{attribute 'GeneratedUsingTerminal: EK1122-0000-0018'}
{attribute addProperty BoxType "EK1122-0000-0018"}
{attribute addProperty Id "Beckhoff_ER6xxxsub_EK1100EK1100_AB5A94672A_0001_ER6001_0002_0016ER6001_B965E9F560A_0002_ER6001_0002_0021ER6001_B965E9F560A_0003_ER6002_0002_0021ER6002_EA7A2404108A_0004_ER6002_0002_0022ER6002_EECF1379108A_0005_ER6002_0002_0023ER6002_EECF1379108"}
{attribute addProperty CRC "2923937941"}
{attribute addProperty Size "446"}
TYPE Beckhoff_ER6xxxEK1122_AE47C095 EXTENDS EK1122_AB5A9467 :
STRUCT
	{attribute addProperty Name "Beckhoff_ER6xxxsub_EK1100"}
	{attribute addProperty PreviousPort "Beckhoff ER6xxxEK1122 : D"}
	Beckhoff_ER6xxxsub_EK1100 : EK1100_AB5A9467;
	{attribute addProperty Name "A_0001_ER6001_0002_0016"}
	{attribute addProperty PreviousPort "Beckhoff ER6xxxsub EK1100 : C"}
	A_0001_ER6001_0002_0016 : ER6001_B965E9F5;
	{attribute addProperty Name "A_0002_ER6001_0002_0021"}
	{attribute addProperty PreviousPort "A_0001(ER6001-0002-0016) : B"}
	A_0002_ER6001_0002_0021 : ER6001_B965E9F5;
	{attribute addProperty Name "A_0003_ER6002_0002_0021"}
	{attribute addProperty PreviousPort "A_0002(ER6001-0002-0021) : B"}
	A_0003_ER6002_0002_0021 : ER6002_EA7A2404;
	{attribute addProperty Name "A_0004_ER6002_0002_0022"}
	{attribute addProperty PreviousPort "A_0003(ER6002-0002-0021) : B"}
	A_0004_ER6002_0002_0022 : ER6002_EECF1379;
	{attribute addProperty Name "A_0005_ER6002_0002_0023"}
	{attribute addProperty PreviousPort "A_0004(ER6002-0002-0022) : B"}
	A_0005_ER6002_0002_0023 : ER6002_EECF1379;
END_STRUCT
END_TYPE

(* stored: Version 1.2.0.0, ProductVersion 3.1.4024.9
   DUT Beckhoff_ER6xxxEK1122_AE47C095: Id {763778fc-5c07-4c25-8f23-a8fd4dcf7a04} *)
